Yaskawa INFORM job: R1_W49-52-A2(90,90)KM-OK.JBI

/JOB
//NAME R1_W49-52-A2(90,90)KM-OK
///FOLDERNAME KRIS-SCIANA
//POS
///NPOS 61,61,0,3,0,0
///TOOL 0
///POSTYPE PULSE
///PULSE
C00000=-67926,8916,-30568,-8968,94185,-35982
C00001=-73499,58572,17801,5922,119515,-36735
C00002=-82155,59631,25834,4037,115644,-40158
C00003=-80395,51171,39276,4532,107387,-38885
C00004=-80395,52450,44312,4468,104952,-38977
C00005=-80395,53073,46462,4444,103953,-39014
C00006=-80223,52302,46352,4478,103616,-38965
C00007=-80395,53073,46462,4444,103953,-39014
C00008=-80980,57364,52471,6246,114422,-44048
C00009=-80818,56142,51092,6326,114628,-43974
C00010=-81202,53511,47267,5198,113721,-44148
C00011=-84530,49317,47350,32123,95915,-39257
C00012=-83989,50344,48476,32187,95568,-39140
C00013=-81922,50742,46211,27432,97419,-37666
C00014=-80391,53692,48530,25002,99085,-36655
C00015=-80390,53383,47546,25040,99491,-36567
C00016=-120616,65183,63772,-6404,94057,-37704
C00017=-120607,45241,41952,-6256,89025,-35963
C00018=-120604,39035,36186,-6272,85483,-35785
C00019=-120616,67167,67875,-6266,92940,-36160
C00020=-120616,67847,69214,3680,92433,-36923
C00021=-120616,66398,68472,3678,92145,-36931
C00022=-120616,67847,69214,3680,92433,-36923
C00023=-120616,66266,65627,3688,93825,-36882
C00024=-120397,14904,9684,-7425,73193,-82165
C00025=-120602,15569,14454,-7481,70601,-82078
C00026=-119669,16188,16486,-7740,69760,-81688
C00027=-120597,13987,13799,-7500,70195,-82051
C00028=-120597,17083,16579,-7505,70076,-82043
C00029=-120603,16134,16269,-7518,69776,-82026
C00030=-120603,16025,16225,-7519,69747,-82024
C00031=-120603,15998,16113,-7515,69807,-82027
C00032=-120602,15557,14411,-7480,70621,-82079
C00033=-120601,14894,9643,-7378,73194,-82238
C00034=-119572,-9619,-19929,-2131,105200,-53554
C00035=-120520,19747,17769,-2437,117887,-54144
C00036=-120609,19829,19332,-2462,117303,-54167
C00037=-120823,-17207,-21082,-2265,101979,-53934
C00038=-120750,-18786,-22608,-2257,102108,-53912
C00039=-120586,-16994,-15120,5410,111704,-56480
C00040=-120586,-17556,-16581,5437,112311,-56451
C00041=-120585,-18321,-20232,5524,114157,-56361
C00042=-120548,-52664,-74582,5146,105241,-56762
C00043=-85553,-41383,-68223,3777,105261,-45062
C00044=-77887,-47932,-44703,-45716,66077,-62645
C00045=-79818,-14659,-13376,-50465,85257,-54730
C00046=-81841,35097,42008,-55452,107604,-42486
C00047=-88972,58431,73291,-49230,109701,-37033
C00048=-91747,59832,78118,-49681,106753,-36840
C00049=-91295,46962,61486,-49875,102611,-50481
C00050=-92289,58805,76923,-49950,106606,-37039
C00051=-92481,61841,80898,-49794,105922,-36756
C00052=-92690,45496,59817,-50360,102045,-50891
C00053=-88308,38208,49129,-51828,100881,-47285
C00054=-88972,58431,73291,-49230,109701,-37033
C00055=-80975,34302,45414,-59271,106254,-42023
C00056=-75646,39754,43353,-59239,111678,-42720
C00057=-74619,29751,20548,-63032,116814,-46507
C00058=-68561,9782,-14722,-63877,106879,-54644
C00059=-39692,-143275,-127218,-62410,73467,-46566
C00060=-1562,-143275,-127218,-62410,38256,61362
BC00000=260492,45975,1075170
BC00001=260492,45975,1075170
BC00002=260492,45975,1075170
BC00003=260942,45747,1075175
BC00004=262985,42394,1075175
BC00005=263802,41053,1075175
BC00006=263802,41053,1075175
BC00007=263802,41053,1075175
BC00008=273014,56662,1053112
BC00009=273014,56662,1053112
BC00010=273014,56662,1053112
BC00011=226713,50923,1053594
BC00012=226713,50923,1053594
BC00013=226713,50923,1053594
BC00014=224965,52413,1060916
BC00015=220596,56139,1075175
BC00016=382321,15,1075175
BC00017=382123,15,1075175
BC00018=382111,15,1075175
BC00019=382123,15,1075175
BC00020=364709,15,1075175
BC00021=364693,15,1075175
BC00022=364709,15,1075175
BC00023=364181,15,1075175
BC00024=398174,15,1075175
BC00025=397708,15,1075175
BC00026=394541,15,1075175
BC00027=397295,15,1075175
BC00028=397295,15,1075175
BC00029=394541,15,1075175
BC00030=392516,15,1075175
BC00031=389763,15,1075175
BC00032=390177,15,1075175
BC00033=391211,15,1075175
BC00034=377915,67012,1075175
BC00035=380277,64457,1075175
BC00036=381221,63434,1075175
BC00037=381221,63434,1075175
BC00038=381221,63434,1075175
BC00039=372122,88746,1075175
BC00040=370917,90471,1075175
BC00041=367904,94782,1075175
BC00042=367904,94782,1075175
BC00043=367904,94782,1075175
BC00044=398174,21672,1075175
BC00045=398174,21672,1075175
BC00046=398174,21672,1075175
BC00047=398174,21672,1075175
BC00048=398174,21672,1075175
BC00049=398172,20735,1075171
BC00050=398174,20734,1075175
BC00051=398174,20734,1075175
BC00052=398172,20735,1075171
BC00053=398172,20735,1075171
BC00054=398174,21672,1075175
BC00055=398174,21672,1075175
BC00056=398174,21672,1075175
BC00057=398174,21672,1075175
BC00058=398174,21672,1075175
BC00059=398174,2824,1075175
BC00060=99602,2824,1075175
///POSTYPE BASE
///RECTAN
///RCONF 0,0,0,0,1,0,0,0,0,0,0,0,0,0,0,0,0,0,0,0,0,0,0,0
P00006=2.006,1.622,-0.565,0.0000,0.0000,0.0000
///RCONF 0,0,0,0,0,0,0,0,0,0,0,0,0,0,0,0,0,0,0,0,0,0,0,0
P00023=-2.957,-4.083,2.762,0.0000,0.0000,0.0000
P00024=-1.466,-0.226,-0.419,0.0000,0.0000,0.0000
//INST
///DATE 2024/09/16 12:17
///ATTR SC,RW
///GROUP1 RB1,BS1
NOP
'r1_W49-52-A2(90,90)(z_reki)
'Path S1175
SFTOF
MOVJ C00000 BC00000 VJ=100.00
MOVJ C00001 BC00001 VJ=100.00
MOVJ C00002 BC00002 VJ=100.00
MOVJ C00003 BC00003 VJ=15.00
MOVJ C00004 BC00004 VJ=10.00
MOVL C00005 BC00005 V=60.0
REFP 3 C00006 BC00006
CALL JOB:SEARCH-R1
SET P024 P006
SFTON P024
MOVL C00007 BC00007 V=60.0
MOVL C00008 BC00008 V=60.0
REFP 3 C00009 BC00009
CALL JOB:SEARCH-R1
SET P024 P006
SFTON P024
MOVL C00010 BC00010 V=60.0
MOVL C00011 BC00011 V=60.0
REFP 3 C00012 BC00012
CALL JOB:SEARCH-R1
SET P024 P006
SFTON P024
MOVL C00013 BC00013 V=100.0
MOVL C00014 BC00014 V=166.7
MOVL C00015 BC00015 V=250.0
'Path S1176
SFTOF
MOVL C00016 BC00016 V=250.0
MOVL C00017 BC00017 V=100.0
REFP 3 C00018 BC00018
CALL JOB:SEARCH-R1
SET P023 P006
SFTON P023
MOVL C00019 BC00019 V=133.3
MOVL C00020 BC00020 V=100.0
REFP 3 C00021 BC00021
CALL JOB:SEARCH-R1
SET P023 P006
SFTON P023
MOVL C00022 BC00022 V=60.0
MOVL C00023 BC00023 V=83.3
'Path W1177
SFTOF
SFTON P023
MOVL C00024 BC00024 V=166.7
MOVL C00025 BC00025 V=166.7
CALL JOB:COFNIJ_DRUT
MOVL C00026 BC00026 V=133.3 PL=0
REFP 1 C00027 BC00027
REFP 2 C00028 BC00028
MACRO1 MJ#(0) ARGF7
ARCON
MOVL C00029 BC00029 V=10.8
MOVL C00030 BC00030 V=10.8
MOVL C00031 BC00031 V=10.8
ARCOF
MOVL C00032 BC00032 V=166.7
MOVL C00033 BC00033 V=166.7
SFTOF
'Path W1178
SFTOF
SFTON P024
MOVJ C00034 BC00034 VJ=15.00
MOVJ C00035 BC00035 VJ=15.00
MOVL C00036 BC00036 V=100.0 PL=0
REFP 1 C00037 BC00037
REFP 2 C00038 BC00038
MACRO1 MJ#(0) ARGF9
ARCON
MOVL C00039 BC00039 V=10.0
ARCOF
MOVL C00040 BC00040 V=100.0
MOVL C00041 BC00041 V=166.7
SFTOF
'Path VIA1213
SFTOF
MOVJ C00042 BC00042 VJ=20.00
'Path VIA1214
SFTOF
MOVJ C00043 BC00043 VJ=100.00
'Path VIA1222
SFTOF
MOVJ C00044 BC00044 VJ=15.00
'Path VIA1221
SFTOF
MOVJ C00045 BC00045 VJ=15.00
'Path VIA1220
SFTOF
MOVJ C00046 BC00046 VJ=10.00
'Path VIA1219
SFTOF
MOVJ C00047 BC00047 VJ=15.00
'Path W1179
SFTOF
SFTON P024
MOVJ C00048 BC00048 VJ=15.00
MOVL C00049 BC00049 V=100.0 PL=0
REFP 1 C00050 BC00050
REFP 2 C00051 BC00051
MACRO1 MJ#(0) ARGF0
MOVL C00052 BC00052 V=10.0
ARCOF
MOVL C00053 BC00053 V=166.7
SFTOF
'Path VIA1215
SFTOF
MOVJ C00054 BC00054 VJ=10.00
'Path VIA1216
SFTOF
MOVJ C00055 BC00055 VJ=10.00
'Path VIA1217
SFTOF
MOVJ C00056 BC00056 VJ=15.00
'Path VIA1218
SFTOF
MOVJ C00057 BC00057 VJ=15.00
MOVJ C00058 BC00058 VJ=100.00
MOVJ C00059 BC00059 VJ=100.00
MOVJ C00060 BC00060 VJ=100.00
END
